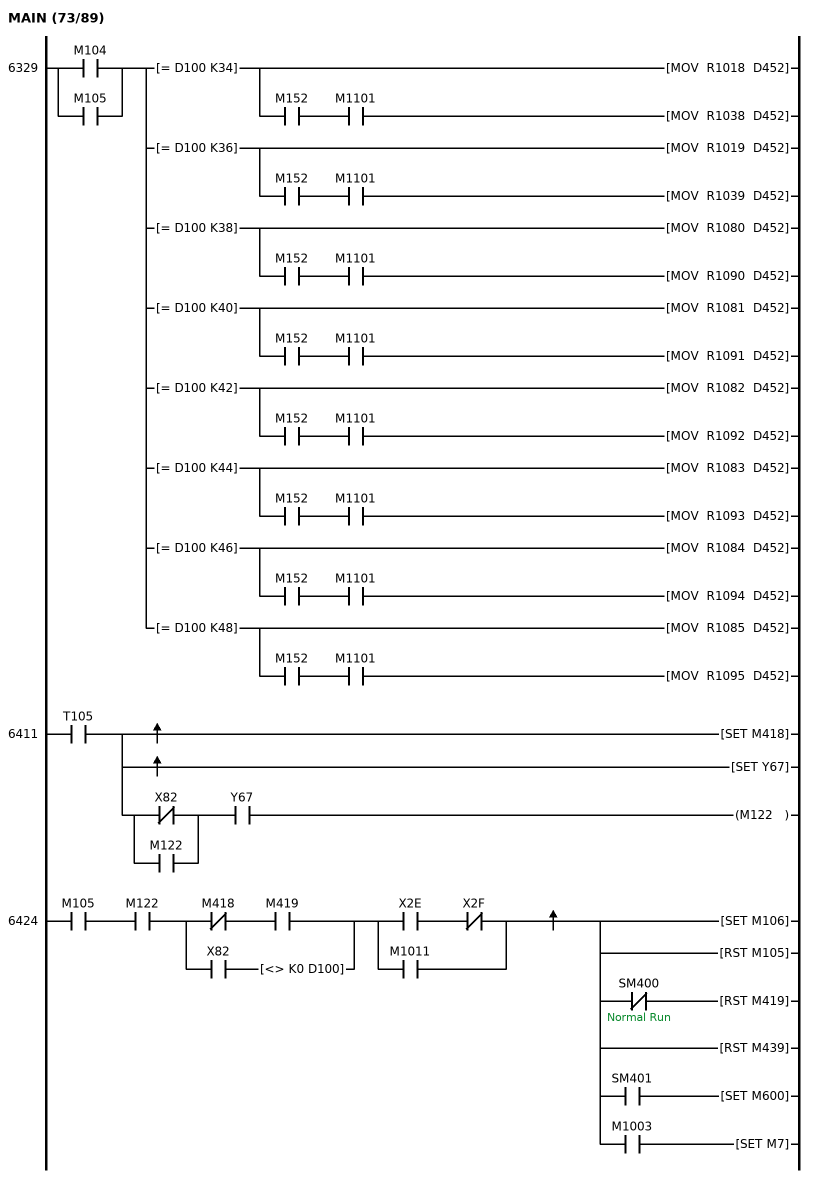
[picture p72: ladder of MAIN, rungs at steps 6329 to 6424]
6329  LD      M104
      OR      M105
      MPS
      AND=    D100 K34
      MOV     R1018 D452
      AND     M152
      AND     M1101
      MOV     R1038 D452
      MRD
      AND=    D100 K36
      MOV     R1019 D452
      AND     M152
      AND     M1101
      MOV     R1039 D452
      MRD
      AND=    D100 K38
      MOV     R1080 D452
      AND     M152
      AND     M1101
      MOV     R1090 D452
      MRD
      AND=    D100 K40
      MOV     R1081 D452
      AND     M152
      AND     M1101
      MOV     R1091 D452
      MRD
      AND=    D100 K42
      MOV     R1082 D452
      AND     M152
      AND     M1101
      MOV     R1092 D452
      MRD
      AND=    D100 K44
      MOV     R1083 D452
      AND     M152
      AND     M1101
      MOV     R1093 D452
      MRD
      AND=    D100 K46
      MOV     R1084 D452
      AND     M152
      AND     M1101
      MOV     R1094 D452
      MPP
      AND=    D100 K48
      MOV     R1085 D452
      AND     M152
      AND     M1101
      MOV     R1095 D452
6411  LD      T105
      MPS
      MEP
      SET     M418
      MRD
      MEP
      SET     Y67
      MPP
      LDI     X82
      OR      M122
      ANB
      AND     Y67
      OUT     M122
6424  LD      M105
      AND     M122
      LDI     M418
      AND     M419
      LD      X82
      AND<>   K0 D100
      ORB
      ANB
      LD      X2E
      ANI     X2F
      OR      M1011
      ANB
      MEP
      SET     M106
      RST     M105
      MPS
      ANI     SM400  ; Normal Run
      RST     M419
      MPP
      RST     M439
      MPS
      AND     SM401
      SET     M600
      MPP
      AND     M1003
      SET     M7
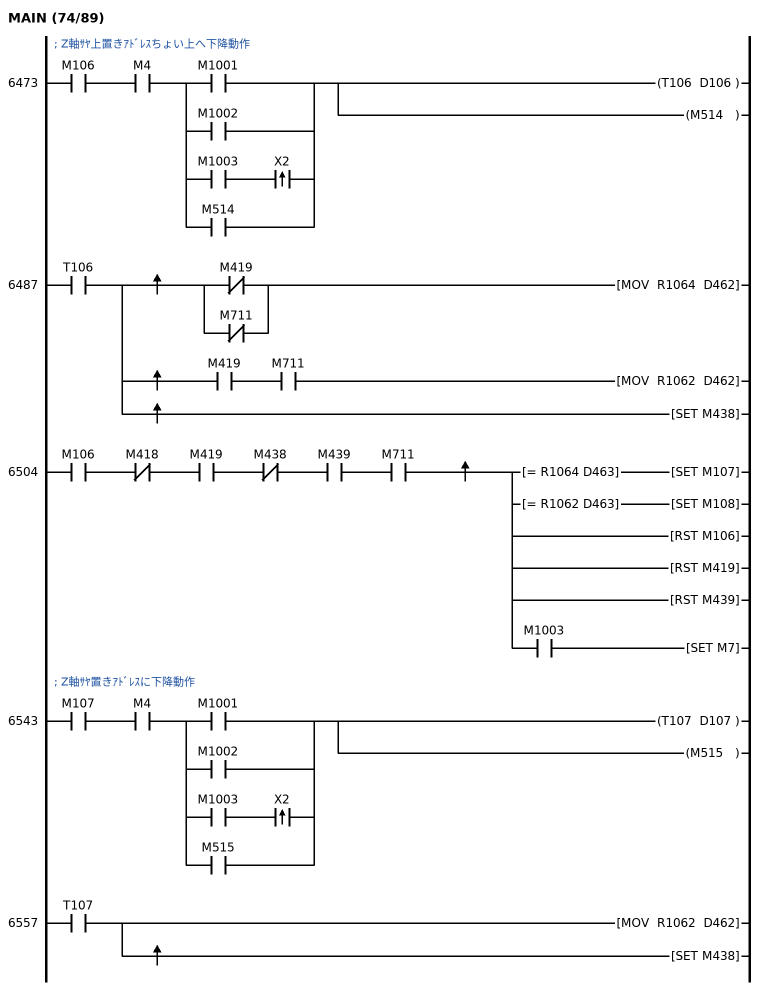
; Z軸ｻﾔ上置きｱﾄﾞﾚｽちょい上へ下降動作
6473  LD      M106
      AND     M4
      LD      M1001
      OR      M1002
      LD      M1003
      ANDP    X2
      ORB
      OR      M514
      ANB
      OUT     T106 D106
      OUT     M514
6487  LD      T106
      MPS
      MEP
      LDI     M419
      ORI     M711
      ANB
      MOV     R1064 D462
      MRD
      MEP
      AND     M419
      AND     M711
      MOV     R1062 D462
      MPP
      MEP
      SET     M438
6504  LD      M106
      ANI     M418
      AND     M419
      ANI     M438
      AND     M439
      AND     M711
      MEP
      MPS
      AND=    R1064 D463
      SET     M107
      MRD
      AND=    R1062 D463
      SET     M108
      MPP
      RST     M106
      RST     M419
      RST     M439
      AND     M1003
      SET     M7
; Z軸ｻﾔ置きｱﾄﾞﾚｽに下降動作
6543  LD      M107
      AND     M4
      LD      M1001
      OR      M1002
      LD      M1003
      ANDP    X2
      ORB
      OR      M515
      ANB
      OUT     T107 D107
      OUT     M515
6557  LD      T107
      MOV     R1062 D462
      MEP
      SET     M438
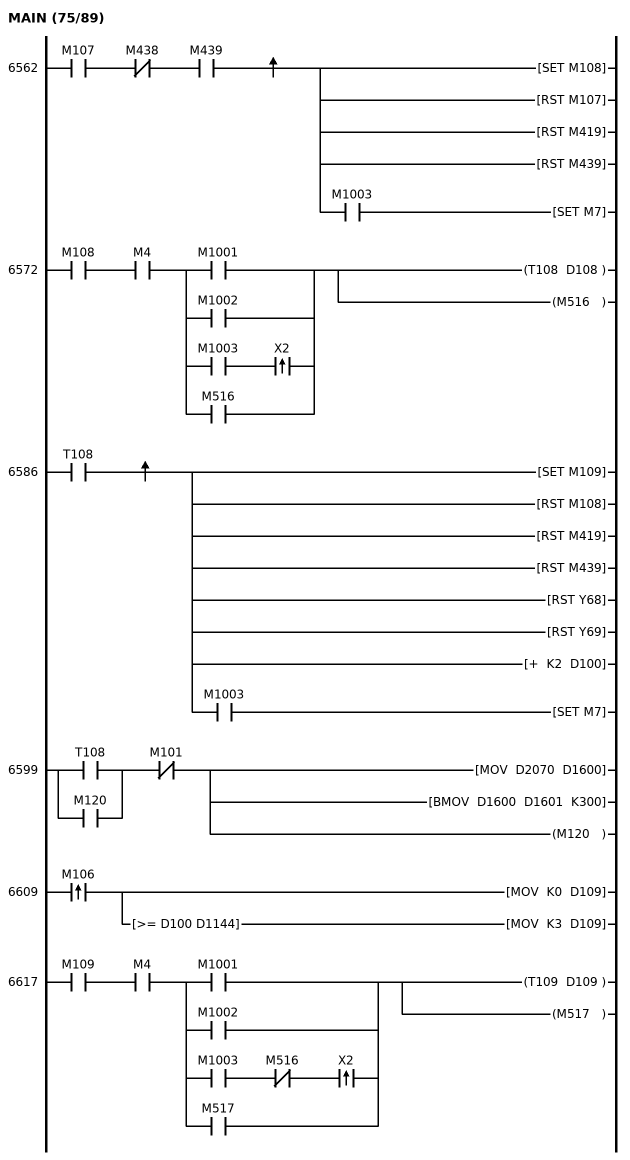
6562  LD      M107
      ANI     M438
      AND     M439
      MEP
      SET     M108
      RST     M107
      RST     M419
      RST     M439
      AND     M1003
      SET     M7
6572  LD      M108
      AND     M4
      LD      M1001
      OR      M1002
      LD      M1003
      ANDP    X2
      ORB
      OR      M516
      ANB
      OUT     T108 D108
      OUT     M516
6586  LD      T108
      MEP
      SET     M109
      RST     M108
      RST     M419
      RST     M439
      RST     Y68
      RST     Y69
      +       K2 D100
      AND     M1003
      SET     M7
6599  LD      T108
      OR      M120
      ANI     M101
      MOV     D2070 D1600
      BMOV    D1600 D1601 K300
      OUT     M120
6609  LDP     M106
      MOV     K0 D109
      AND>=   D100 D1144
      MOV     K3 D109
6617  LD      M109
      AND     M4
      LD      M1001
      OR      M1002
      LD      M1003
      ANI     M516
      ANDP    X2
      ORB
      OR      M517
      ANB
      OUT     T109 D109
      OUT     M517
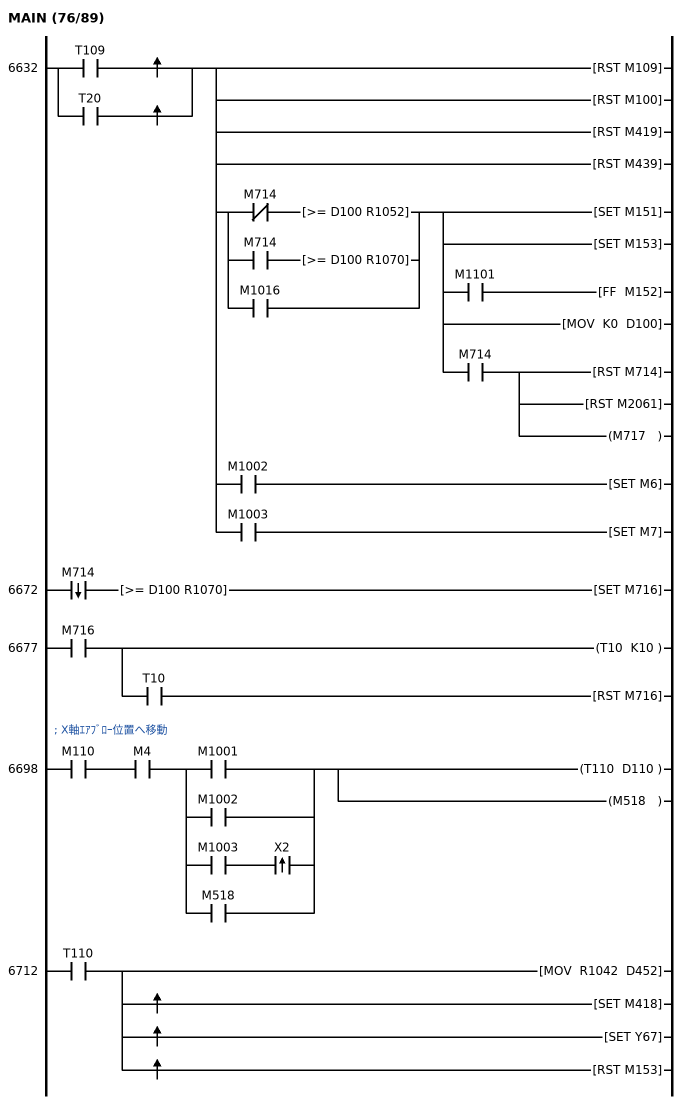
6632  LD      T109
      MEP
      LD      T20
      MEP
      ORB
      RST     M109
      RST     M100
      RST     M419
      RST     M439
      MPS
      LDI     M714
      AND>=   D100 R1052
      LD      M714
      AND>=   D100 R1070
      ORB
      OR      M1016
      ANB
      SET     M151
      SET     M153
      MPS
      AND     M1101
      FF      M152
      MPP
      MOV     K0 D100
      AND     M714
      RST     M714
      RST     M2061
      OUT     M717
      MRD
      AND     M1002
      SET     M6
      MPP
      AND     M1003
      SET     M7
6672  LDF     M714
      AND>=   D100 R1070
      SET     M716
6677  LD      M716
      OUT     T10 K10
      AND     T10
      RST     M716
; X軸ｴｱﾌﾞﾛｰ位置へ移動
6698  LD      M110
      AND     M4
      LD      M1001
      OR      M1002
      LD      M1003
      ANDP    X2
      ORB
      OR      M518
      ANB
      OUT     T110 D110
      OUT     M518
6712  LD      T110
      MOV     R1042 D452
      MPS
      MEP
      SET     M418
      MRD
      MEP
      SET     Y67
      MPP
      MEP
      RST     M153
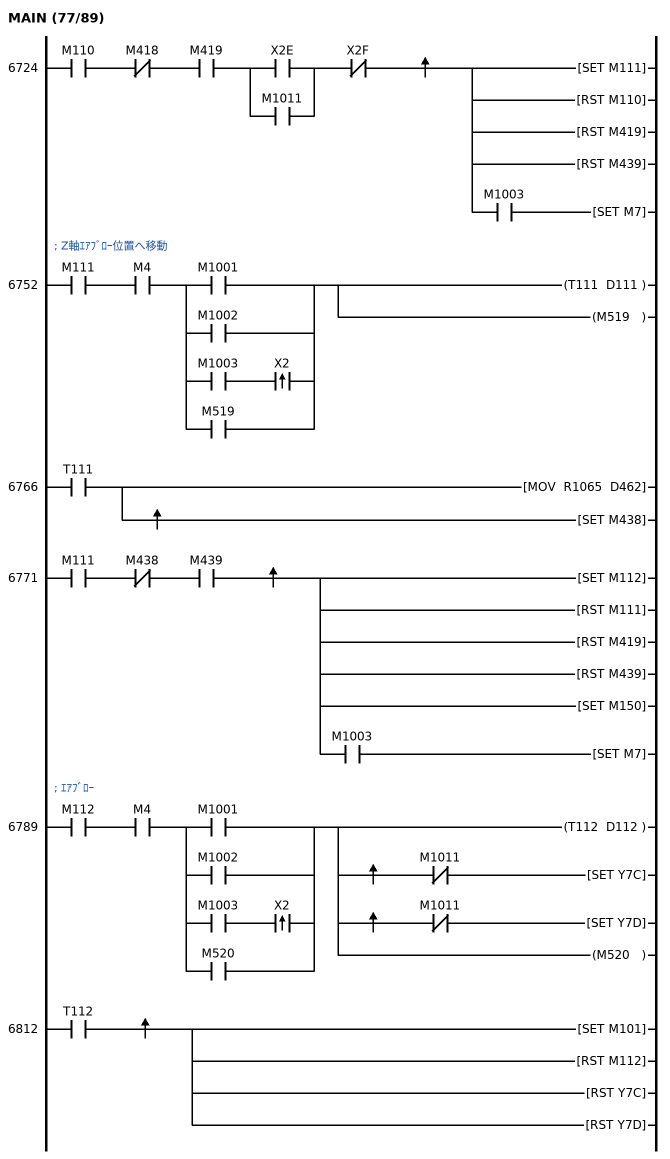
6724  LD      M110
      ANI     M418
      AND     M419
      LD      X2E
      OR      M1011
      ANB
      ANI     X2F
      MEP
      SET     M111
      RST     M110
      RST     M419
      RST     M439
      AND     M1003
      SET     M7
; Z軸ｴｱﾌﾞﾛｰ位置へ移動
6752  LD      M111
      AND     M4
      LD      M1001
      OR      M1002
      LD      M1003
      ANDP    X2
      ORB
      OR      M519
      ANB
      OUT     T111 D111
      OUT     M519
6766  LD      T111
      MOV     R1065 D462
      MEP
      SET     M438
6771  LD      M111
      ANI     M438
      AND     M439
      MEP
      SET     M112
      RST     M111
      RST     M419
      RST     M439
      SET     M150
      AND     M1003
      SET     M7
; ｴｱﾌﾞﾛｰ
6789  LD      M112
      AND     M4
      LD      M1001
      OR      M1002
      LD      M1003
      ANDP    X2
      ORB
      OR      M520
      ANB
      OUT     T112 D112
      MPS
      MEP
      ANI     M1011
      SET     Y7C
      MRD
      MEP
      ANI     M1011
      SET     Y7D
      MPP
      OUT     M520
6812  LD      T112
      MEP
      SET     M101
      RST     M112
      RST     Y7C
      RST     Y7D
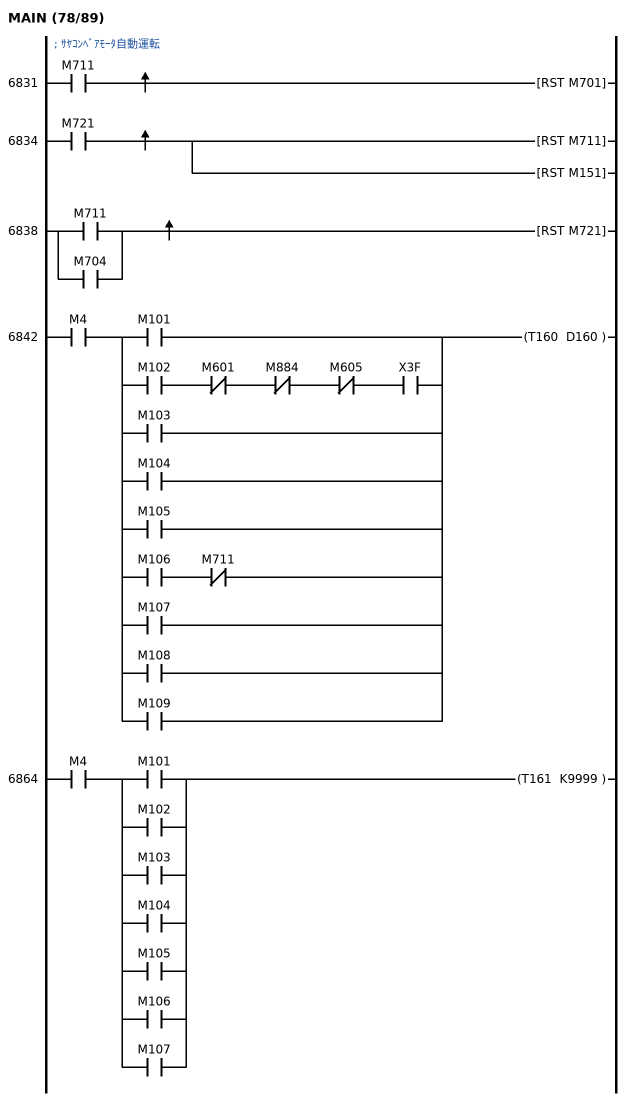
; ｻﾔｺﾝﾍﾞｱﾓｰﾀ自動運転
6831  LD      M711
      MEP
      RST     M701
6834  LD      M721
      MEP
      RST     M711
      RST     M151
6838  LD      M711
      OR      M704
      MEP
      RST     M721
6842  LD      M4
      LD      M101
      LD      M102
      ANI     M601
      ANI     M884
      ANI     M605
      AND     X3F
      ORB
      OR      M103
      OR      M104
      OR      M105
      LD      M106
      ANI     M711
      ORB
      OR      M107
      OR      M108
      OR      M109
      ANB
      OUT     T160 D160
6864  LD      M4
      LD      M101
      OR      M102
      OR      M103
      OR      M104
      OR      M105
      OR      M106
      OR      M107
      ANB
      OUT     T161 K9999
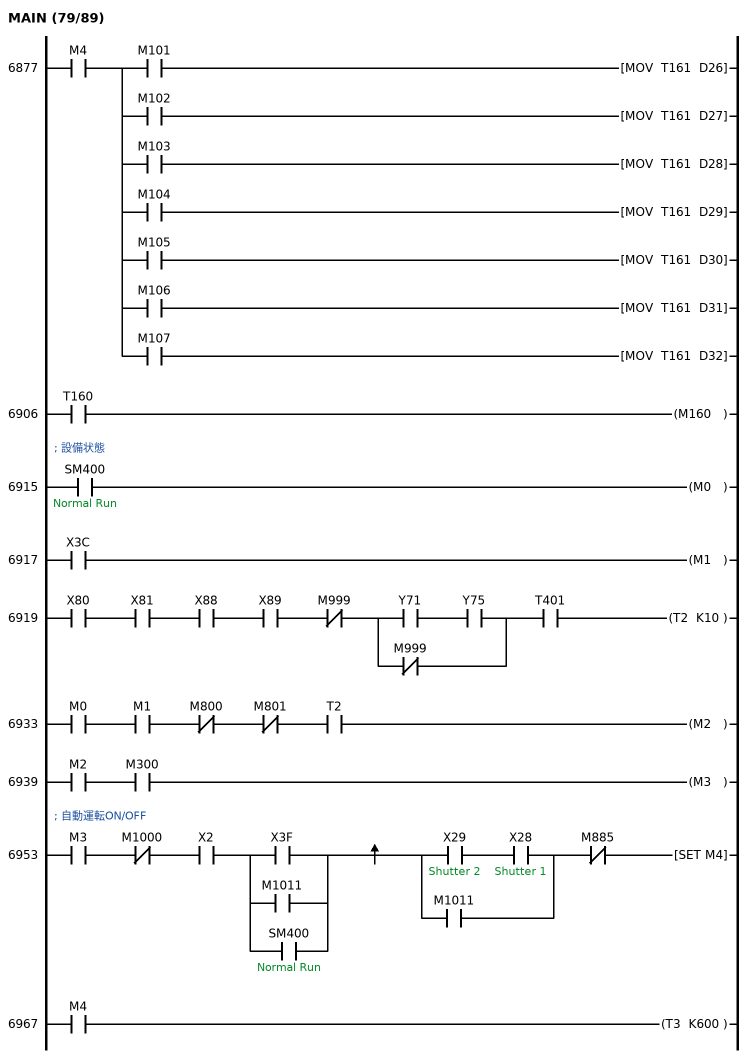
6877  LD      M4
      MPS
      AND     M101
      MOV     T161 D26
      MRD
      AND     M102
      MOV     T161 D27
      MRD
      AND     M103
      MOV     T161 D28
      MRD
      AND     M104
      MOV     T161 D29
      MRD
      AND     M105
      MOV     T161 D30
      MRD
      AND     M106
      MOV     T161 D31
      MPP
      AND     M107
      MOV     T161 D32
6906  LD      T160
      OUT     M160
; 設備状態
; 
6915  LD      SM400  ; Normal Run
      OUT     M0
6917  LD      X3C
      OUT     M1
6919  LD      X80
      AND     X81
      AND     X88
      AND     X89
      ANI     M999
      LD      Y71
      AND     Y75
      ORI     M999
      ANB
      AND     T401
      OUT     T2 K10
6933  LD      M0
      AND     M1
      ANI     M800
      ANI     M801
      AND     T2
      OUT     M2
6939  LD      M2
      AND     M300
      OUT     M3
; 自動運転ON/OFF
6953  LD      M3
      ANI     M1000
      AND     X2
      LD      X3F
      OR      M1011
      OR      SM400  ; Normal Run
      ANB
      MEP
      LD      X29  ; Shutter 2
      AND     X28  ; Shutter 1
      OR      M1011
      ANB
      ANI     M885
      SET     M4
6967  LD      M4
      OUT     T3 K600
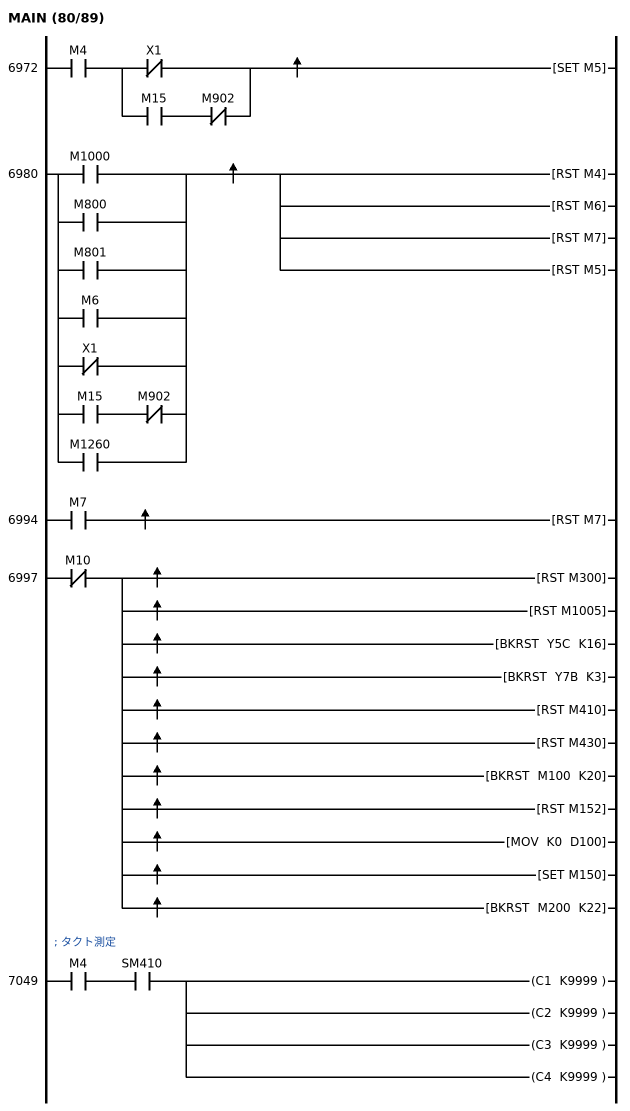
6972  LD      M4
      LDI     X1
      LD      M15
      ANI     M902
      ORB
      ANB
      MEP
      SET     M5
6980  LD      M1000
      OR      M800
      OR      M801
      OR      M6
      ORI     X1
      LD      M15
      ANI     M902
      ORB
      OR      M1260
      MEP
      RST     M4
      RST     M6
      RST     M7
      RST     M5
6994  LD      M7
      MEP
      RST     M7
6997  LDI     M10
      MPS
      MEP
      RST     M300
      MRD
      MEP
      RST     M1005
      MRD
      MEP
      BKRST   Y5C K16
      MRD
      MEP
      BKRST   Y7B K3
      MRD
      MEP
      RST     M410
      MRD
      MEP
      RST     M430
      MRD
      MEP
      BKRST   M100 K20
      MRD
      MEP
      RST     M152
      MRD
      MEP
      MOV     K0 D100
      MRD
      MEP
      SET     M150
      MPP
      MEP
      BKRST   M200 K22
; タクト測定
7049  LD      M4
      AND     SM410
      OUT     C1 K9999
      OUT     C2 K9999
      OUT     C3 K9999
      OUT     C4 K9999
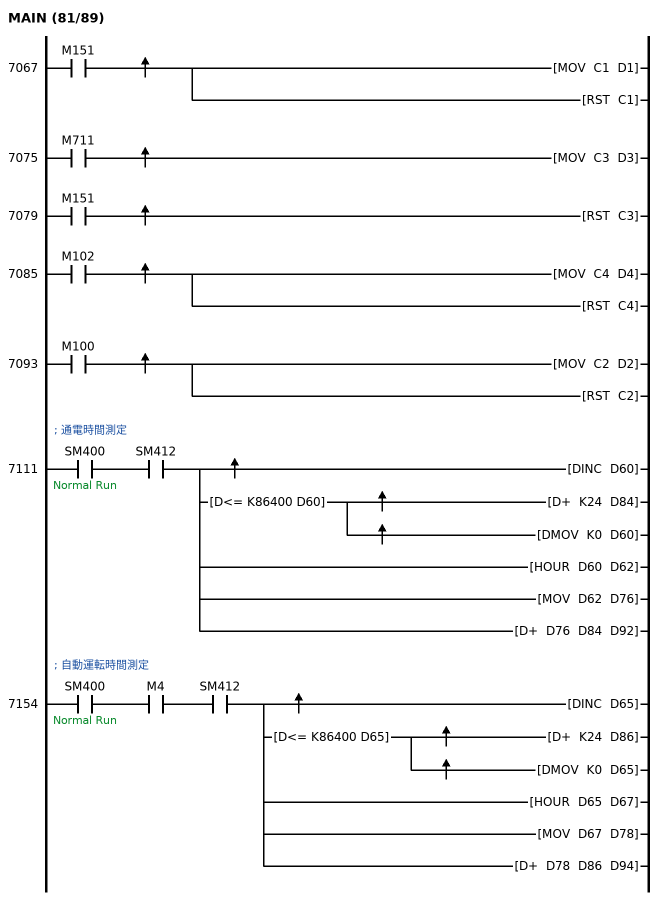
7067  LD      M151
      MEP
      MOV     C1 D1
      RST     C1
7075  LD      M711
      MEP
      MOV     C3 D3
7079  LD      M151
      MEP
      RST     C3
7085  LD      M102
      MEP
      MOV     C4 D4
      RST     C4
7093  LD      M100
      MEP
      MOV     C2 D2
      RST     C2
; 通電時間測定
7111  LD      SM400  ; Normal Run
      AND     SM412
      MPS
      MEP
      DINC    D60
      MRD
      ANDD<=  K86400 D60
      MPS
      MEP
      D+      K24 D84
      MPP
      MEP
      DMOV    K0 D60
      MPP
      HOUR    D60 D62
      MOV     D62 D76
      D+      D76 D84 D92
; 自動運転時間測定
7154  LD      SM400  ; Normal Run
      AND     M4
      AND     SM412
      MPS
      MEP
      DINC    D65
      MRD
      ANDD<=  K86400 D65
      MPS
      MEP
      D+      K24 D86
      MPP
      MEP
      DMOV    K0 D65
      MPP
      HOUR    D65 D67
      MOV     D67 D78
      D+      D78 D86 D94
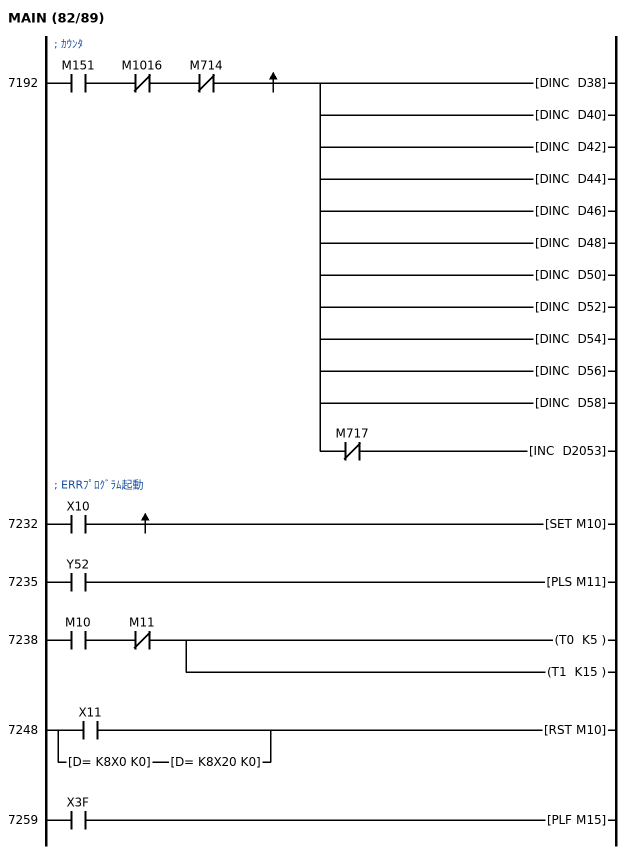
; ｶｳﾝﾀ
7192  LD      M151
      ANI     M1016
      ANI     M714
      MEP
      DINC    D38
      DINC    D40
      DINC    D42
      DINC    D44
      DINC    D46
      DINC    D48
      DINC    D50
      DINC    D52
      DINC    D54
      DINC    D56
      DINC    D58
      ANI     M717
      INC     D2053
; ERRﾌﾟﾛｸﾞﾗﾑ起動
7232  LD      X10
      MEP
      SET     M10
7235  LD      Y52
      PLS     M11
7238  LD      M10
      ANI     M11
      OUT     T0 K5
      OUT     T1 K15
7248  LD      X11
      LDD=    K8X0 K0
      ANDD=   K8X20 K0
      ORB
      RST     M10
7259  LD      X3F
      PLF     M15
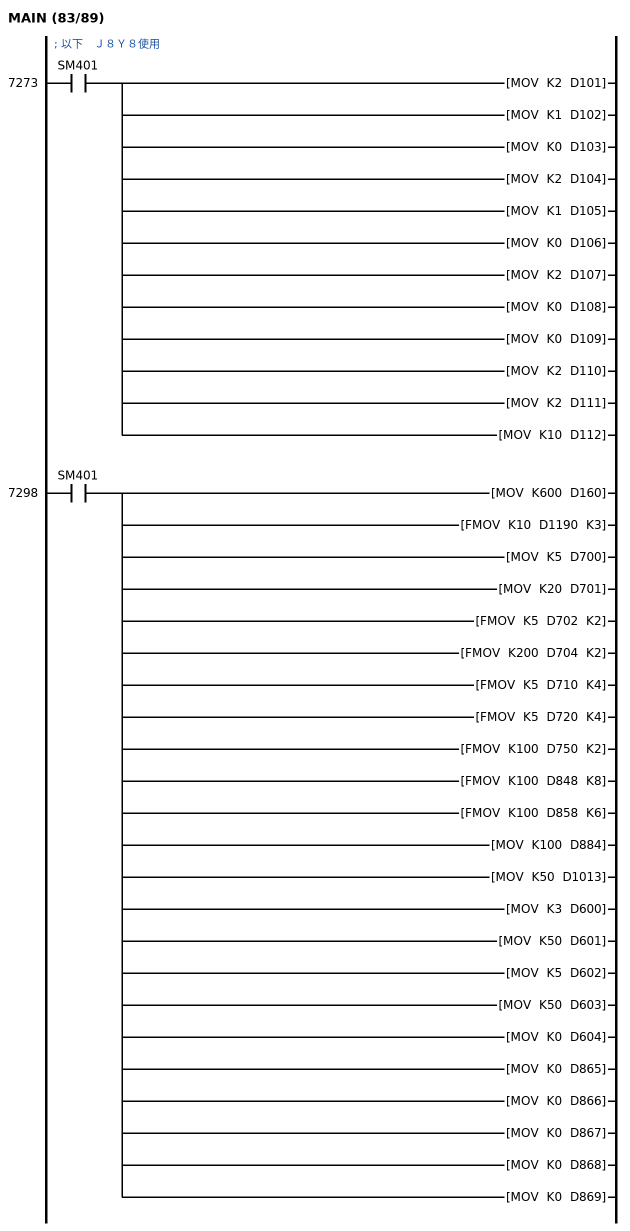
; 以下　Ｊ８Ｙ８使用
7273  LD      SM401
      MOV     K2 D101
      MOV     K1 D102
      MOV     K0 D103
      MOV     K2 D104
      MOV     K1 D105
      MOV     K0 D106
      MOV     K2 D107
      MOV     K0 D108
      MOV     K0 D109
      MOV     K2 D110
      MOV     K2 D111
      MOV     K10 D112
7298  LD      SM401
      MOV     K600 D160
      FMOV    K10 D1190 K3
      MOV     K5 D700
      MOV     K20 D701
      FMOV    K5 D702 K2
      FMOV    K200 D704 K2
      FMOV    K5 D710 K4
      FMOV    K5 D720 K4
      FMOV    K100 D750 K2
      FMOV    K100 D848 K8
      FMOV    K100 D858 K6
      MOV     K100 D884
      MOV     K50 D1013
      MOV     K3 D600
      MOV     K50 D601
      MOV     K5 D602
      MOV     K50 D603
      MOV     K0 D604
      MOV     K0 D865
      MOV     K0 D866
      MOV     K0 D867
      MOV     K0 D868
      MOV     K0 D869
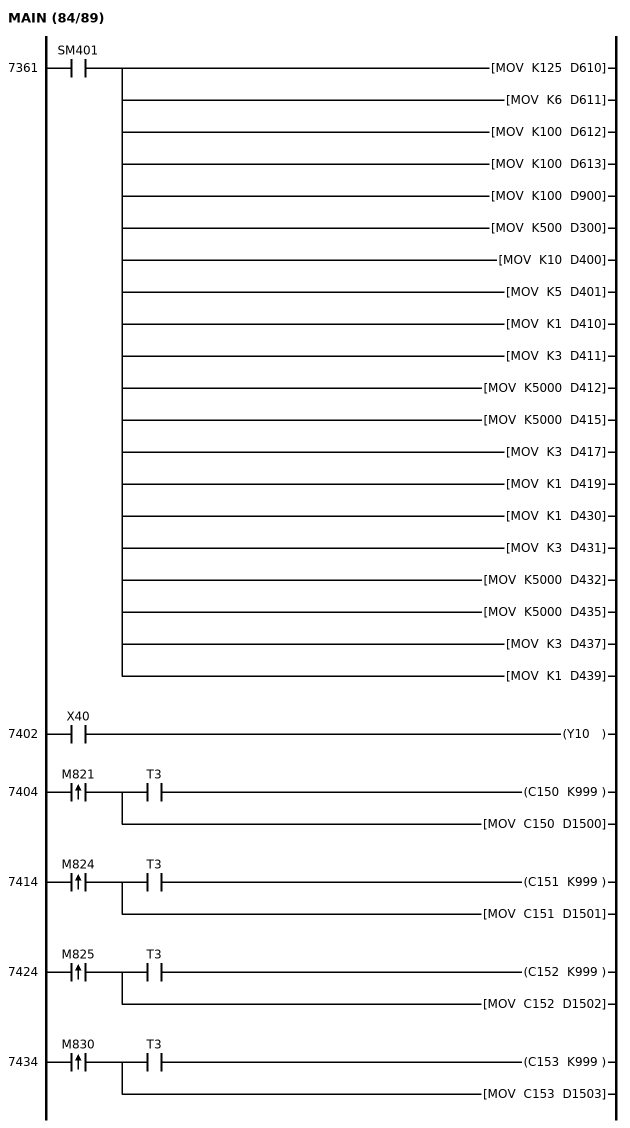
7361  LD      SM401
      MOV     K125 D610
      MOV     K6 D611
      MOV     K100 D612
      MOV     K100 D613
      MOV     K100 D900
      MOV     K500 D300
      MOV     K10 D400
      MOV     K5 D401
      MOV     K1 D410
      MOV     K3 D411
      MOV     K5000 D412
      MOV     K5000 D415
      MOV     K3 D417
      MOV     K1 D419
      MOV     K1 D430
      MOV     K3 D431
      MOV     K5000 D432
      MOV     K5000 D435
      MOV     K3 D437
      MOV     K1 D439
7402  LD      X40
      OUT     Y10
7404  LDP     M821
      MPS
      AND     T3
      OUT     C150 K999
      MPP
      MOV     C150 D1500
7414  LDP     M824
      MPS
      AND     T3
      OUT     C151 K999
      MPP
      MOV     C151 D1501
7424  LDP     M825
      MPS
      AND     T3
      OUT     C152 K999
      MPP
      MOV     C152 D1502
7434  LDP     M830
      MPS
      AND     T3
      OUT     C153 K999
      MPP
      MOV     C153 D1503
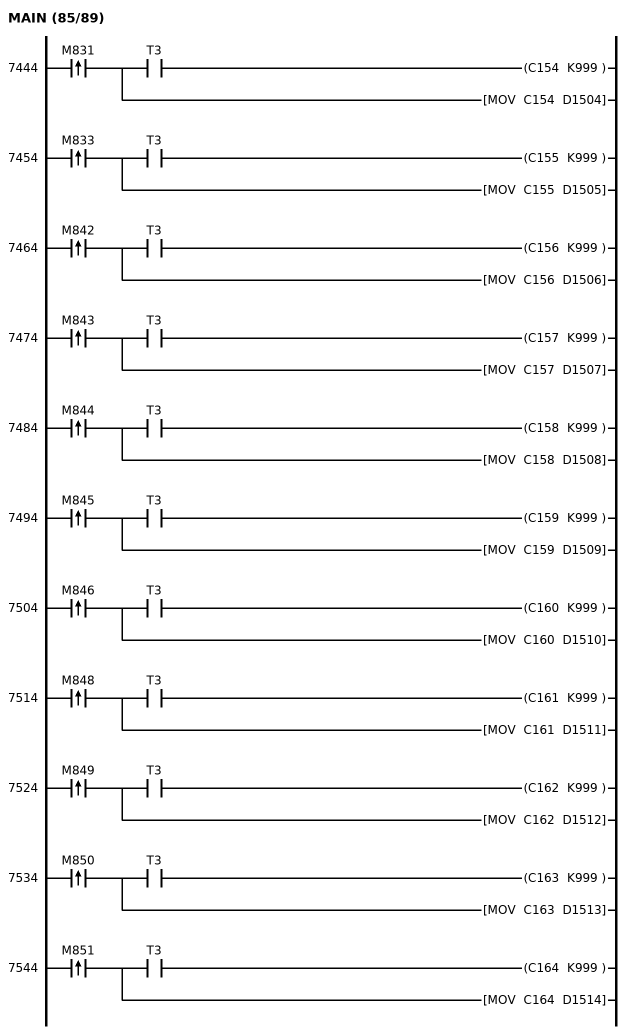
7444  LDP     M831
      MPS
      AND     T3
      OUT     C154 K999
      MPP
      MOV     C154 D1504
7454  LDP     M833
      MPS
      AND     T3
      OUT     C155 K999
      MPP
      MOV     C155 D1505
7464  LDP     M842
      MPS
      AND     T3
      OUT     C156 K999
      MPP
      MOV     C156 D1506
7474  LDP     M843
      MPS
      AND     T3
      OUT     C157 K999
      MPP
      MOV     C157 D1507
7484  LDP     M844
      MPS
      AND     T3
      OUT     C158 K999
      MPP
      MOV     C158 D1508
7494  LDP     M845
      MPS
      AND     T3
      OUT     C159 K999
      MPP
      MOV     C159 D1509
7504  LDP     M846
      MPS
      AND     T3
      OUT     C160 K999
      MPP
      MOV     C160 D1510
7514  LDP     M848
      MPS
      AND     T3
      OUT     C161 K999
      MPP
      MOV     C161 D1511
7524  LDP     M849
      MPS
      AND     T3
      OUT     C162 K999
      MPP
      MOV     C162 D1512
7534  LDP     M850
      MPS
      AND     T3
      OUT     C163 K999
      MPP
      MOV     C163 D1513
7544  LDP     M851
      MPS
      AND     T3
      OUT     C164 K999
      MPP
      MOV     C164 D1514
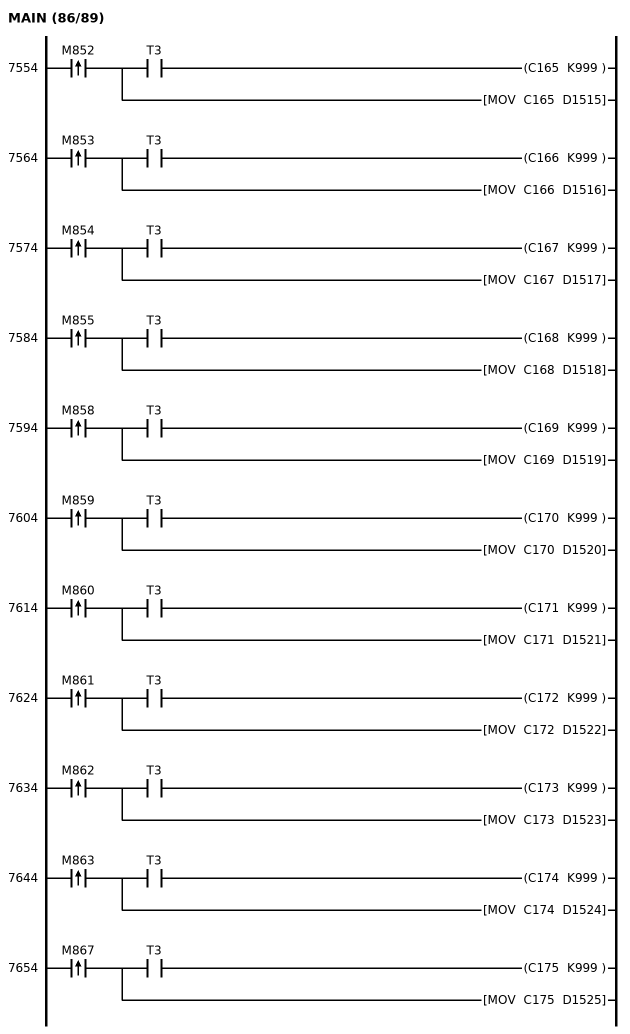
7554  LDP     M852
      MPS
      AND     T3
      OUT     C165 K999
      MPP
      MOV     C165 D1515
7564  LDP     M853
      MPS
      AND     T3
      OUT     C166 K999
      MPP
      MOV     C166 D1516
7574  LDP     M854
      MPS
      AND     T3
      OUT     C167 K999
      MPP
      MOV     C167 D1517
7584  LDP     M855
      MPS
      AND     T3
      OUT     C168 K999
      MPP
      MOV     C168 D1518
7594  LDP     M858
      MPS
      AND     T3
      OUT     C169 K999
      MPP
      MOV     C169 D1519
7604  LDP     M859
      MPS
      AND     T3
      OUT     C170 K999
      MPP
      MOV     C170 D1520
7614  LDP     M860
      MPS
      AND     T3
      OUT     C171 K999
      MPP
      MOV     C171 D1521
7624  LDP     M861
      MPS
      AND     T3
      OUT     C172 K999
      MPP
      MOV     C172 D1522
7634  LDP     M862
      MPS
      AND     T3
      OUT     C173 K999
      MPP
      MOV     C173 D1523
7644  LDP     M863
      MPS
      AND     T3
      OUT     C174 K999
      MPP
      MOV     C174 D1524
7654  LDP     M867
      MPS
      AND     T3
      OUT     C175 K999
      MPP
      MOV     C175 D1525
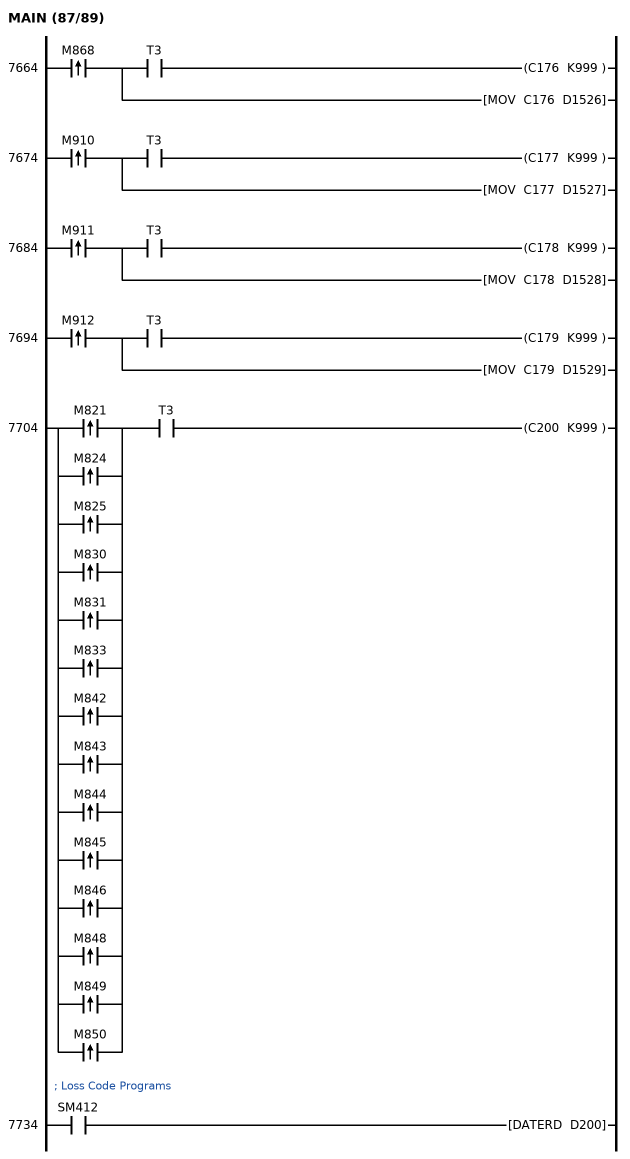
7664  LDP     M868
      MPS
      AND     T3
      OUT     C176 K999
      MPP
      MOV     C176 D1526
7674  LDP     M910
      MPS
      AND     T3
      OUT     C177 K999
      MPP
      MOV     C177 D1527
7684  LDP     M911
      MPS
      AND     T3
      OUT     C178 K999
      MPP
      MOV     C178 D1528
7694  LDP     M912
      MPS
      AND     T3
      OUT     C179 K999
      MPP
      MOV     C179 D1529
7704  LDP     M821
      ORP     M824
      ORP     M825
      ORP     M830
      ORP     M831
      ORP     M833
      ORP     M842
      ORP     M843
      ORP     M844
      ORP     M845
      ORP     M846
      ORP     M848
      ORP     M849
      ORP     M850
      AND     T3
      OUT     C200 K999
; Loss Code Programs
7734  LD      SM412
      DATERD  D200
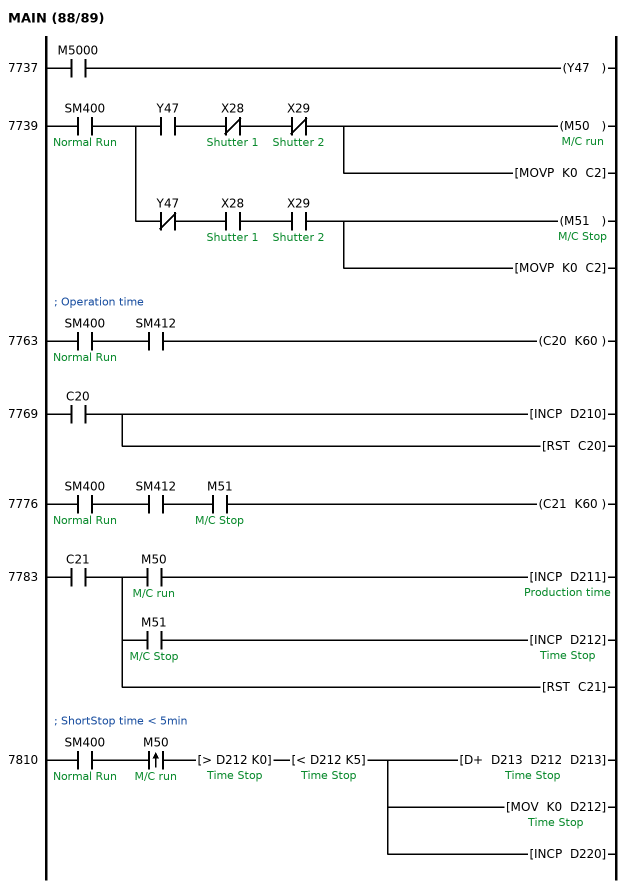
7737  LD      M5000
      OUT     Y47
7739  LD      SM400  ; Normal Run
      MPS
      AND     Y47
      ANI     X28  ; Shutter 1
      ANI     X29  ; Shutter 2
      OUT     M50  ; M/C run
      MOVP    K0 C2
      MPP
      ANI     Y47
      AND     X28  ; Shutter 1
      AND     X29  ; Shutter 2
      OUT     M51  ; M/C Stop
      MOVP    K0 C2
; Operation time
7763  LD      SM400  ; Normal Run
      AND     SM412
      OUT     C20 K60
7769  LD      C20
      INCP    D210
      RST     C20
7776  LD      SM400  ; Normal Run
      AND     SM412
      AND     M51  ; M/C Stop
      OUT     C21 K60
7783  LD      C21
      MPS
      AND     M50  ; M/C run
      INCP    D211  ; Production time
      MRD
      AND     M51  ; M/C Stop
      INCP    D212  ; Time Stop
      MPP
      RST     C21
; ShortStop time < 5min
7810  LD      SM400  ; Normal Run
      ANDP    M50  ; M/C run
      AND>    D212 K0  ; Time Stop
      AND<    D212 K5  ; Time Stop
      D+      D213 D212 D213
      MOV     K0 D212
      INCP    D220
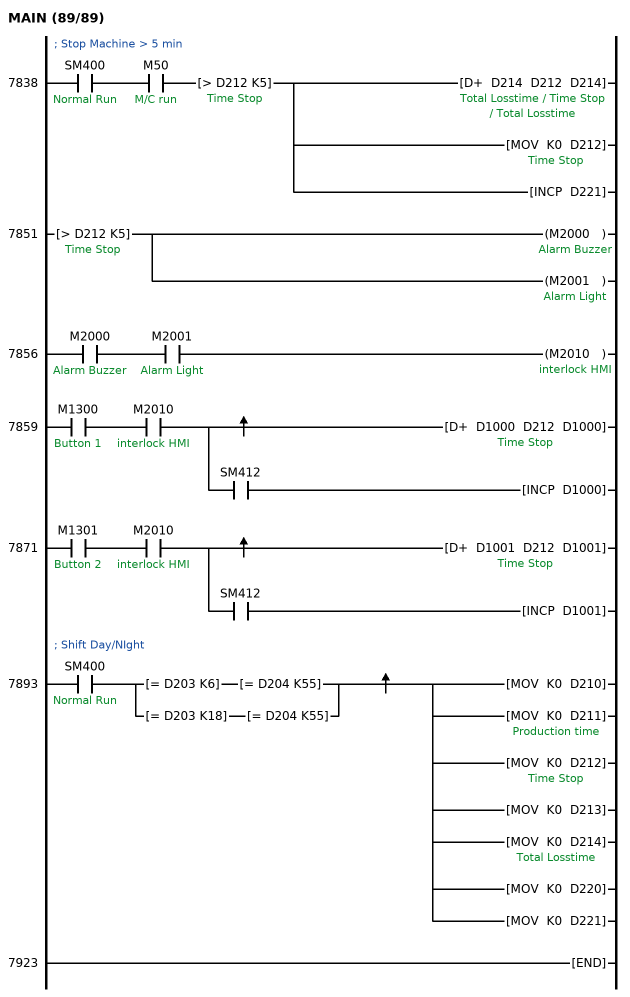
; Stop Machine > 5 min
7838  LD      SM400  ; Normal Run
      AND     M50  ; M/C run
      AND>    D212 K5  ; Time Stop
      D+      D214 D212 D214  ; Total Losstime
      MOV     K0 D212
      INCP    D221
7851  LD>     D212 K5  ; Time Stop
      OUT     M2000  ; Alarm Buzzer
      OUT     M2001  ; Alarm Light
7856  LD      M2000  ; Alarm Buzzer
      AND     M2001  ; Alarm Light
      OUT     M2010  ; interlock HMI
7859  LD      M1300  ; Button 1
      AND     M2010  ; interlock HMI
      MPS
      MEP
      D+      D1000 D212 D1000
      MPP
      AND     SM412
      INCP    D1000
7871  LD      M1301  ; Button 2
      AND     M2010  ; interlock HMI
      MPS
      MEP
      D+      D1001 D212 D1001
      MPP
      AND     SM412
      INCP    D1001
; Shift Day/NIght
7893  LD      SM400  ; Normal Run
      LD=     D203 K6
      AND=    D204 K55
      LD=     D203 K18
      AND=    D204 K55
      ORB
      ANB
      MEP
      MOV     K0 D210
      MOV     K0 D211
      MOV     K0 D212
      MOV     K0 D213
      MOV     K0 D214
      MOV     K0 D220
      MOV     K0 D221
7923  END
END_PROGRAM
